{attribute 'Tc2GvlVarNames'}
{attribute 'strict'}
//Tipologia Falda
TYPE e_Tipo_Falda :
(
	NOT_DEFINED				:= -1,
	FALDA_CARTONE 			:= 1, (* Falde di Cartone *)
	FALDA_POLISTIROLO 		:= 2, (* Falde di Polistirolo *)
	MISTO					:= 999
);
END_TYPE
//  NOT_DEFINED = '-1'

(* stored: Version 1.1.0.1, ProductVersion 3.1.4024.11
   EnumerationTextList e_Tipo_Falda: Id {29a0f01f-73ec-464b-9876-d5b998ab3931} *)
